TYPE ST_EM_Sts :
	STRUCT
		CurrentTable : UDINT;
	END_STRUCT
END_TYPE

(* stored: Version 1.1.0.1, ProductVersion 3.1.4024.12
   DUT ST_EM_Sts: Id {e4a0fc70-885f-422b-9d51-c72c49bc5155} *)
